(* PLC project 117_1_V0.5.project, CODESYS CODESYS V3.5 SP17 Patch 3 *)
(* stored: creationDateTime 1970-01-01T00:00:00, modificationDateTime 2026-06-16T22:51:19.9979415 *)

TYPE PID_DIAGNOSTIC_UDT : STRUCT
  Error : REAL;
  PreviousError : REAL;
  Proportional : REAL;
  Integral : REAL;
  Differential : REAL;
  Status : PID_STATUS_UDT;
  Direction : PID_DIRECTION_UDT;
  Kp : REAL;
  Ki : REAL;
  Kd : REAL;
  Ts : TIME;
  MinOut : REAL;
  MaxOut : REAL;
END_STRUCT;
END_TYPE
